INTERFACE iDelta

METHOD ExecuteRoute : BOOL
VAR_INPUT
END_VAR
END_METHOD

METHOD MoveDirectTo : BOOL
VAR_INPUT
END_VAR
END_METHOD

METHOD MoveX : BOOL
VAR_INPUT
END_VAR
END_METHOD

METHOD MoveY : BOOL
VAR_INPUT
END_VAR
END_METHOD

METHOD MoveZ : BOOL
VAR_INPUT
END_VAR
END_METHOD

METHOD ReturnHome : BOOL
VAR_INPUT
END_VAR
END_METHOD

METHOD SetAcceleration : BOOL
VAR_INPUT
	Acceleration	: LREAL;
END_VAR
END_METHOD

METHOD SetDeceleration : BOOL
VAR_INPUT
END_VAR
END_METHOD

METHOD SetJerk : BOOL
VAR_INPUT
END_VAR
END_METHOD

METHOD SetVelocity : BOOL
VAR_INPUT
END_VAR
END_METHOD

METHOD TraverseAtHeightTo : BOOL
VAR_INPUT
END_VAR
END_METHOD

END_INTERFACE

(* stored: Version 1.1.0.1, ProductVersion 3.1.4024.11
   Itf iDelta: Id {b1c10141-048b-4915-a2fa-88aacf371a42}
   Folder Methods: Id {c034fcca-b79b-4a07-919e-0aa436878a14}
   Folder Properties: Id {7f0fa4d5-5926-4280-a4f1-3aa8c199ef0b}
   Method ExecuteRoute: Id {372bd43e-1964-4819-9927-4766da54fadd}
   Method MoveDirectTo: Id {d2077d88-8c04-4ac5-86df-9bb4f09b9f7b}
   Method MoveX: Id {0b33ef1c-3cf0-449b-9029-982734f1bb91}
   Method MoveY: Id {68ed6926-92dc-4a76-a033-5e0f4cbdece1}
   Method MoveZ: Id {65ef6f9b-1600-4494-8dce-d06a52da1d70}
   Method ReturnHome: Id {cf0bd24f-f8dd-4060-9275-9cd153896c40}
   Method SetAcceleration: Id {59eed68b-e3b3-46b8-8d4d-101f238de2b4}
   Method SetDeceleration: Id {92e76549-e495-400b-8163-d30d797cd585}
   Method SetJerk: Id {f358d58c-b7b1-4086-9187-de99b7eafcec}
   Method SetVelocity: Id {50a06832-0f68-4d62-8c3e-aa920e16ea8b}
   Method TraverseAtHeightTo: Id {5f0f7064-58f5-43fc-ac8f-ef9da33cd706} *)
